Fanuc KAREL source: kb00102.KL

-- PROVISIONAL review KL for V940-1; original PC SHA256 e4f8efacbf1d657dcfa8f2e8361eaa6664ef94f98d292af325509a2a52e326a4
-- Incomplete behavior may be omitted. Consult companion uncertainty JSON. Do not deploy.
PROGRAM KB00102
%NOLOCKGROUP
BEGIN
  -- V9_ZERO_TABLE_METADATA_HINT layout=0002_ascii; no indexed target words; source/name/runtime held
  -- UNRESOLVED_PC offsets 5-12; opcodes 9D,23
  -- UNRESOLVED_PC offsets 17-26; opcodes 3F,75
  -- UNRESOLVED_PC offsets 31-38; opcodes 9D,23
  -- UNRESOLVED_PC offsets 43-50; opcodes 9D,23
  -- UNRESOLVED_PC offsets 55-62; opcodes 9D,23
  -- UNRESOLVED_PC offsets 67-74; opcodes 9D,23
  -- UNRESOLVED_PC offsets 79-86; opcodes 9D,23
  -- UNRESOLVED_PC offsets 91-98; opcodes 9D,23
  -- UNRESOLVED_PC offsets 103-110; opcodes 9D,23
  -- UNRESOLVED_PC offsets 115-124; opcodes 3F,75
  -- UNRESOLVED_PC offsets 129-136; opcodes 9D,23
  -- UNRESOLVED_PC offsets 141-215; opcodes 27,22,22,2A,22,22,22,22,22,22,22,22,2A,22,31
  -- UNRESOLVED_PC offsets 220-224; opcodes 7F
END KB00102
